Staubli VAL3: resetControlSocket.pgx

program resetControlSocket(sio& x_UdpSocket, bool& x_bError)
begin
  // Non-blocking socket
  sioCtrl(x_UdpSocket, "timeout", -1)
  // Linux EoL ('\n')
  sioCtrl(x_UdpSocket, "endOfString", 10)
  // Clear buffer
  clearBuffer(x_UdpSocket)

  x_bError = false
end
